(* PLC project Programme MGS_2-07_refactorJOY.project, CODESYS CODESYS V3.5 SP19 Patch 1 *)
(* stored: creationDateTime 2026-06-29T23:37:40.3099964, modificationDateTime 2026-06-29T22:49:33.424 *)

FUNCTION_BLOCK FB_Joystick
  VAR_INPUT
    Enable : BOOL;  (* Active la logique *)
    Reset : BOOL;  (* Acquittement défaut *)
    SafeStop : BOOL;  (* Arrêt sûr forcé *)
    SafetyOk : BOOL;  (* Conditions globales OK *)
    CanOnline : BOOL;  (* État présence nœud CAN *)
    CanOperational : BOOL;  (* Mode esclave CANopen actif *)
    RawX : INT;  (* Valeur brute axe X *)
    RawY : INT;  (* Valeur brute axe Y *)
    RawButton : BOOL;  (* État brut bouton *)
    Calibrate : BOOL;  (* Demande de recalage neutre *)
    InvertX : BOOL := FALSE;
    InvertY : BOOL := FALSE;
    Deadband : REAL := 5;
    FilterTime : TIME := TIME#100ms;
    AccelRate : REAL := 50;
    DecelRate : REAL := 150;
  END_VAR
  VAR_OUTPUT
    Ready : BOOL;  (* Prêt à commuter *)
    Busy : BOOL;  (* Traitement en cours *)
    Done : BOOL;  (* Données valides dispo *)
    Error : BOOL;  (* Présence anomalie *)
    ErrorId : WORD;  (* Code d'erreur *)
    AxisCmdX : ST_AxisCmd;  (* Sortie normalisée X *)
    AxisCmdY : ST_AxisCmd;  (* Sortie normalisée Y *)
    Button : BOOL;  (* Bouton filtré *)
    NeutralXAct : INT;  (* Point neutre X actuel pour IHM/Test *)
    NeutralYAct : INT;  (* Point neutre Y actuel pour IHM/Test *)
  END_VAR
  VAR RETAIN
    NeutralXMem : INT := 5000;  (* Mémoire persistante X *)
    NeutralYMem : INT := 5000;  (* Mémoire persistante Y *)
  END_VAR
  VAR
    CycleTimeCalc : FB_CycleTime;
    ScaleX : FB_AxisScale;
    ScaleY : FB_AxisScale;
    FilterX : FB_Filter_PT1;
    FilterY : FB_Filter_PT1;
    RampX : FB_Ramp;
    RampY : FB_Ramp;
    LastCalibrate : BOOL;
  END_VAR

            // 🛑 1. GATE (Sécurités et coupures prioritaires)
IF NOT Enable OR SafeStop OR NOT CanOnline OR NOT CanOperational THEN
    Ready := FALSE; Busy := FALSE; Done := FALSE;
    AxisCmdX.Enable := FALSE; AxisCmdX.Start := FALSE; AxisCmdX.SpeedRef := 0.0; AxisCmdX.Direction := 0; AxisCmdX.SafetyOk := FALSE;
    AxisCmdY.Enable := FALSE; AxisCmdY.Start := FALSE; AxisCmdY.SpeedRef := 0.0; AxisCmdY.Direction := 0; AxisCmdY.SafetyOk := FALSE;
    Button := FALSE;
    NeutralXAct := NeutralXMem;
    NeutralYAct := NeutralYMem;
    RETURN;
END_IF;

Ready := TRUE; Busy := TRUE;

// 🔑 2. RESET DÉFAUT
IF Reset AND Error THEN
    Error := FALSE; ErrorId := 16#0000;
END_IF;

// 📥 3. ACQUISITION TIMING & BOUTON
CycleTimeCalc();
Button := RawButton;

// 🎯 4. CALIBRATION DYNAMIQUE (Zone RETAIN)
IF Calibrate AND NOT LastCalibrate THEN
    IF RawX >= 2000 AND RawX <= 8000 AND RawY >= 2000 AND RawY <= 8000 THEN
        NeutralXMem := RawX;
        NeutralYMem := RawY;
    ELSE
        Error := TRUE; ErrorId := 16#0003;
    END_IF;
END_IF;
LastCalibrate := Calibrate;

// 🕹️ 5. PIPELINE TRAITEMENT — AXE X
ScaleX(RawIn := RawX, Neutral := NeutralXMem, Deadband := Deadband);

IF InvertX THEN
    FilterX(ValueIn := -ScaleX.OutPct, TimeConst := FilterTime, CycleTimeS := CycleTimeCalc.CycleTimeS);
ELSE
    FilterX(ValueIn := ScaleX.OutPct, TimeConst := FilterTime, CycleTimeS := CycleTimeCalc.CycleTimeS);
END_IF;

RampX(Target := FilterX.ValueOut, AccelRate := AccelRate, DecelRate := DecelRate, CycleTimeS := CycleTimeCalc.CycleTimeS);

// Mapping Sortie Standardisée Axe X
AxisCmdX.Enable := TRUE;
AxisCmdX.SpeedRef := ABS(RampX.Current);
AxisCmdX.Start := (AxisCmdX.SpeedRef > 0.1);
AxisCmdX.SafetyOk := SafetyOk;

IF RampX.Current > 0.1 THEN     AxisCmdX.Direction := 1;
ELSIF RampX.Current < -0.1 THEN AxisCmdX.Direction := -1;
ELSE AxisCmdX.Direction := 0;   AxisCmdX.SpeedRef := 0.0;
END_IF;

// 🕹️ 6. PIPELINE TRAITEMENT — AXE Y
ScaleY(RawIn := RawY, Neutral := NeutralYMem, Deadband := Deadband);

IF InvertY THEN
    FilterY(ValueIn := -ScaleY.OutPct, TimeConst := FilterTime, CycleTimeS := CycleTimeCalc.CycleTimeS);
ELSE
    FilterY(ValueIn := ScaleY.OutPct, TimeConst := FilterTime, CycleTimeS := CycleTimeCalc.CycleTimeS);
END_IF;

RampY(Target := FilterY.ValueOut, AccelRate := AccelRate, DecelRate := DecelRate, CycleTimeS := CycleTimeCalc.CycleTimeS);

// Mapping Sortie Standardisée Axe Y
AxisCmdY.Enable := TRUE;
AxisCmdY.SpeedRef := ABS(RampY.Current);
AxisCmdY.Start := (AxisCmdY.SpeedRef > 0.1);
AxisCmdY.SafetyOk := SafetyOk;

IF RampY.Current > 0.1 THEN     AxisCmdY.Direction := 1;
ELSIF RampY.Current < -0.1 THEN AxisCmdY.Direction := -1;
ELSE AxisCmdY.Direction := 0;   AxisCmdY.SpeedRef := 0.0;
END_IF;

// 📤 7. VALIDATION DES SORTIES ÉTAT
NeutralXAct := NeutralXMem;
NeutralYAct := NeutralYMem;
Done := NOT Error;
          
END_FUNCTION_BLOCK
